INTERFACE I_Command

METHOD execute : BOOL
VAR_INPUT
END_VAR
END_METHOD

END_INTERFACE

(* stored: Version 1.1.0.1
   Itf I_Command: Id {b78fe57d-cd6e-47d3-a847-eb9ff7b43455}
   Method execute: Id {4871210d-9105-44da-a0c4-4c8528dfd71c} *)
